(*
SPDX-FileCopyrightText: © 2026 Oleksandr Tiutyk <trofimich@gmail.com>
SPDX-License-Identifier: MIT
License: https://opensource.org/license/mit
*)

(*!
<summary>Represents exception diagnostics with task-owned cloning.</summary>
<description>
Dynamic copies are explicitly registered by Clone after construction; plain __NEW does not transfer ownership
to the task manager.
</description>
*)

{attribute 'no_explicit_call' := 'do not call this function block directly'}
{attribute 'enable_dynamic_creation'}
FUNCTION_BLOCK DemoException EXTENDS TOF_Core.GeneralException IMPLEMENTS IDemoException
VAR_STAT
	//! <summary>Class name shared by all instances of this function block.</summary>
	{attribute 'hide'} 
	_ClassName : STRING := __POUNAME();
END_VAR
VAR
	{attribute 'hide'} 
	_IsCritical : BOOL;	
END_VAR

{attribute 'monitoring' := 'call'}
PROPERTY ClassName : REFERENCE TO STRING
GET
ClassName REF= _ClassName;
END_GET
END_PROPERTY

(*!
<summary>Creates a task-owned copy of this exception and its diagnostic payload.</summary>
<description>
Registers the newly constructed instance before copying payload, outside FB_init. Registration failure
releases the unregistered instance and raises a terminal error; copy failure leaves the registered instance
owned by the task manager for cleanup. Custom overrides must follow the same ownership sequence. The returned
reference is borrowed until task cleanup and must not be deleted by the caller.
</description>
*)
METHOD Clone : TOF_Core.IObject
VAR
	exceptionClone : POINTER TO DemoException;
END_VAR
exceptionClone := __NEW(DemoException);

IF exceptionClone = 0 THEN
	TOF_Core.DynamicMemoryManager.RaiseAllocationFailure();
END_IF

TOF_Core.DynamicMemoryManager.RegisterAutoDisposedObject(autoDisposedObject := exceptionClone^);

exceptionClone^.CopyGeneralFields(sourceException := THIS^);
exceptionClone^.IsCritical := _IsCritical;

Clone := exceptionClone^;
END_METHOD

{attribute 'monitoring' := 'call'}
PROPERTY IsCritical : BOOL
GET
IsCritical := _IsCritical;
END_GET
SET // INTERNAL
_IsCritical := IsCritical;
END_SET
END_PROPERTY

{attribute 'monitoring' := 'call'}
PROPERTY NamespaceName : REFERENCE TO STRING
GET
NamespaceName REF= CurrentNamespace.Name;
END_GET
END_PROPERTY

{attribute 'monitoring' := 'call'}
PROPERTY SelfSize : ULINT
GET
SelfSize := XSIZEOF(THIS^);
END_GET
END_PROPERTY

METHOD Throw
VAR_INPUT
	sourceNamespaceName : STRING;
	sourceClassName : STRING;
	sourcePOUName : STRING;
	sourcePosition : STRING;
	isCritical : BOOL;
END_VAR
VAR_IN_OUT CONSTANT
	message : STRING(255);
END_VAR
VAR
	errorMessage : TOF_Core.ERROR_MESSAGE;
END_VAR
_IsCritical := isCritical;

errorMessage := TO_WSTRING(message);

InternalThrow(
	sourceNamespaceName := sourceNamespaceName,
	sourceClassName := sourceClassName,
	sourcePOUName := sourcePOUName,
	sourcePosition := sourcePosition,
	message := errorMessage,
	errorCode := 0,
	innerException := 0
);
END_METHOD

END_FUNCTION_BLOCK

(* stored: Version 1.1.0.1
   POU DemoException: Id {adc8ba1f-b7dc-4ef4-bc68-4f768efa6feb}, SpecialFunc None
   Property ClassName: Id {5c1d72c0-0bd5-4561-8624-e06b4c278b7a}
   Get Get: Id {2af1a41a-d563-45d5-a27a-d9b0604010a3}
   Method Clone: Id {10a3c882-0aae-4a71-8f8c-e40ec80da357}
   Property IsCritical: Id {44c25764-c19c-42ab-813d-47bc781ed2d0}
   Get Get: Id {42cde1da-3e2b-4077-bf48-69f6b2b3e916}
   Set Set: Id {e7d9d481-9287-461c-adeb-3dfa764d874f}
   Property NamespaceName: Id {0d97f348-4c22-4ff3-a42a-ea32e8b20cca}
   Get Get: Id {04a1fff0-a864-4ced-a0a8-84b07f5dc442}
   Property SelfSize: Id {717bf6fc-834d-4c14-a6e9-71f3441879c9}
   Get Get: Id {6cc747b7-a5a5-47c9-b7d7-830bd5bf7812}
   Method Throw: Id {79b3f44d-92d7-4159-b6fc-ab05b70abedf} *)
